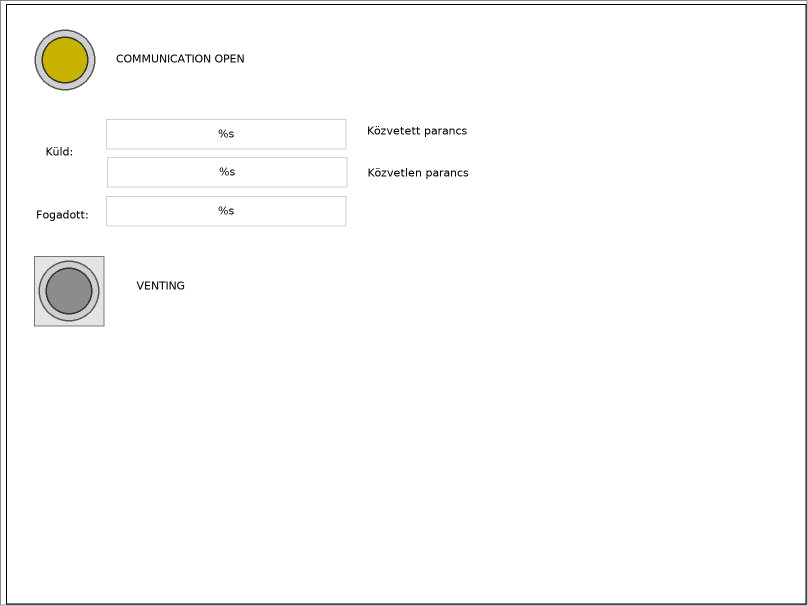
VISUALIZATION Laser  // 808x606
    Rectangle (6,4 800x600)
    Textfield (106,119 240x30), "%s", text variable: Laser.s_InCommand
        OnMouseClick: write Laser.s_InCommand via VisuDialogs.Keypad
    Textfield (106,196 240x30), "%s", text variable: Laser.sLaserReceived
    Lamp1 (30,25 70x70), variable: GVL.bLaserCommOpen, style: Lamp-Lamp1-Yellow
    Label (106,44 149x30), "COMMUNICATION OPEN"
    Label (31,137 57x30), "Küld:"
    Label (30,200 65x30), "Fogadott:"
    PushSwitch (34,256 70x70), variable: AUTOMATA.bElszivasBe, behaviour: TOGGLE, style: Switch-PushSwitch-Gray
    Label (127,271 68x30), "VENTING"
    Label (360,116 114x30), "Közvetett parancs"
    Label (361,158 114x30), "Közvetlen parancs"
    Textfield (107,157 240x30), "%s", text variable: Laser.sLaserSend
        OnMouseClick: write Laser.sLaserSend via VisuDialogs.Keypad
END_VISUALIZATION

(* stored: Version 1.1.0.1, ProductVersion 3.1.4024.11
   Visu Laser: Id {43535a7f-0f93-42b7-ba69-7f766a5ebde1} *)
